(* IEC 61131-3 sources: RL_MAR/experiments/comparison/autoplc/results/gpt-4o_20260511_211137/med_89, 1 file *)

(* ---- med_89_1.st ---- *)
FUNCTION_BLOCK SoilTestingDeviceControl
VAR_INPUT
    StartButton : BOOL; (* Input for starting the testing process *)
    SoilSampleDetected : BOOL; (* Input for detecting soil sample *)
END_VAR
VAR_OUTPUT
    NutrientPump : BOOL; (* Output to control nutrient pump *)
    pHAdjustmentPump : BOOL; (* Output to control pH adjustment pump *)
END_VAR
VAR
    pHSensorValue : REAL; (* Simulated pH sensor value *)
    NutrientSensorValue : REAL; (* Simulated nutrient sensor value *)
    TestingStatus : INT; (* Status: 0=Idle, 1=Testing, 2=Completed *)
    NutrientThreshold : REAL := 0.7; (* Nutrient level threshold for analysis *)
    pHThreshold : REAL := 6.5; (* pH level threshold for analysis *)
END_VAR

(* Initialization *)
IF TestingStatus = 0 THEN
    pHSensorValue := 7.0;
    NutrientSensorValue := 0.5;
END_IF

(* Start/Testing Logic *)
IF StartButton AND (TestingStatus = 0) THEN
    TestingStatus := 1;
    NutrientPump := TRUE;
    pHAdjustmentPump := TRUE;
END_IF

(* Sample Detection and Analysis *)
IF (TestingStatus = 1) THEN
    IF SoilSampleDetected THEN
        IF (NutrientSensorValue >= NutrientThreshold) AND (pHSensorValue <= pHThreshold) THEN
            TestingStatus := 2;
            NutrientPump := FALSE;
            pHAdjustmentPump := FALSE;
        END_IF
    END_IF

    (* Simulated Sensor Value Updates *)
    NutrientSensorValue := NutrientSensorValue + 0.1;
    IF NutrientSensorValue > 0.9 THEN
        NutrientSensorValue := 0.9;
    END_IF

    pHSensorValue := pHSensorValue - 0.5;
    IF pHSensorValue < 4.0 THEN
        pHSensorValue := 4.0;
    END_IF
END_IF

END_FUNCTION_BLOCK
